TYPE ST_ProcessCylinder_CMD :
STRUCT
	
	ExtendCylinder1				: BOOL;		
	RetractCylinder1			: BOOL;		
	ExtendCylinder2				: BOOL;		
	RetractCylinder2			: BOOL;	
	
END_STRUCT
END_TYPE

(* stored: Version 1.1.0.1, ProductVersion 3.1.4024.13
   DUT ST_ProcessCylinder_CMD: Id {be788ca4-1f59-4430-b468-666609eaa6c5} *)
